// TIA Portal V19 export
TYPE "IF_TA2502"
TITLE = TA2502
// DEVICEID : 466
//  VENDOR : ifm electronic gmbh
//  DATE: 27.09.2021 
// 
//  Comment : Interface TA2502
   STRUCT
      StandardStructure : Struct
         Header : Struct
            NumberParameter : Int := 17;   // Number of device parameters (Device Identification + Device Parameter)
            AdressParamDownLoad : Int := 20;   // Start adress for ParamDownload signals in this struct
            AdressDeviceIndent : Int := 44;   // Start adress for Device Identification Parameters in this struct
            AdressApplicSpez : Int := 700;   // Start adress ApplicationSpezificTag
            AdressDeviceParam : Int := 782;   // Start adress for Device Parameters in this Area
            AdressKommando : Int := 942;   // Start adress for Device Commandos
            NumberCommandos : Int := 5;   // Number of Commandos of the device
            Spare01 : Int;   // spare
            Spare02 : Int;   // spare
            Spare03 : Int;   // spare
         END_STRUCT;
         Paramdownload : Struct
            ParamDownLoadStart : Struct   // Parameter Download Start (Only if master and device are V1.1)
               BlockStat : DWord;   // function block status
               IOLStat : DWord;   // IO-Link Status
            END_STRUCT;
            ParamDownLoadEnd : Struct   // Parameter Download End (Only if master and device are V1.1)
               BlockStat : DWord;   // function block status
               IOLStat : DWord;   // IO-Link Status
            END_STRUCT;
            ParamDownLoadStore : Struct   // Parameter Download Store (Only if master and device are V1.1)
               BlockStat : DWord;   // function block status
               IOLStat : DWord;   // IO-Link Status
            END_STRUCT;
         END_STRUCT;
         DeviceIndentification : Struct   // device indentification parameter
            V_VendorName : Struct   // Vendor Name
               Text : String[64];
               Index : Int := 16;   // parameter index
               Subindex : Int;   // parameter subindex
               Length : Int := 19;   // parameter length in BYTE for writing
               BlockStat : DWord;   // function block status
               IOLStat : DWord;   // IO-Link Status
               RelRead : Bool := TRUE;   // reading release
               RelWrite : Bool;   // writing release
            END_STRUCT;
            V_VendorText : Struct   // Vendor Text
               Text : String[64];
               Index : Int := 17;   // parameter index
               Subindex : Int;   // parameter subindex
               Length : Int := 11;   // parameter length in BYTE for writing
               BlockStat : DWord;   // function block status
               IOLStat : DWord;   // IO-Link Status
               RelRead : Bool := TRUE;   // reading release
               RelWrite : Bool;   // writing release
            END_STRUCT;
            V_ProductName : Struct   // Product Name
               Text : String[64];
               Index : Int := 18;   // parameter index
               Subindex : Int;   // parameter subindex
               Length : Int := 6;   // parameter length in BYTE for writing
               BlockStat : DWord;   // function block status
               IOLStat : DWord;   // IO-Link Status
               RelRead : Bool := TRUE;   // reading release
               RelWrite : Bool;   // writing release
            END_STRUCT;
            V_ProductID : Struct   // Product ID
               Text : String[64];
               Index : Int := 19;   // parameter index
               Subindex : Int;   // parameter subindex
               Length : Int := 6;   // parameter length in BYTE for writing
               BlockStat : DWord;   // function block status
               IOLStat : DWord;   // IO-Link Status
               RelRead : Bool := TRUE;   // reading release
               RelWrite : Bool;   // writing release
            END_STRUCT;
            V_ProductText : Struct   // Product Text
               Text : String[64];
               Index : Int := 20;   // parameter index
               Subindex : Int;   // parameter subindex
               Length : Int := 23;   // parameter length in BYTE for writing
               BlockStat : DWord;   // function block status
               IOLStat : DWord;   // IO-Link Status
               RelRead : Bool := TRUE;   // reading release
               RelWrite : Bool;   // writing release
            END_STRUCT;
            V_SerialNumber : Struct   // Serial Number
               Text : String[64];
               Index : Int := 21;   // parameter index
               Subindex : Int;   // parameter subindex
               Length : Int := 12;   // parameter length in BYTE for writing
               BlockStat : DWord;   // function block status
               IOLStat : DWord;   // IO-Link Status
               RelRead : Bool := TRUE;   // reading release
               RelWrite : Bool;   // writing release
            END_STRUCT;
            V_HardwareRevision : Struct   // Hardware Version
               Text : String[64];
               Index : Int := 22;   // parameter index
               Subindex : Int;   // parameter subindex
               Length : Int := 2;   // parameter length in BYTE for writing
               BlockStat : DWord;   // function block status
               IOLStat : DWord;   // IO-Link Status
               RelRead : Bool := TRUE;   // reading release
               RelWrite : Bool;   // writing release
            END_STRUCT;
            V_FirmwareRevision : Struct   // Firmware Version
               Text : String[64];
               Index : Int := 23;   // parameter index
               Subindex : Int;   // parameter subindex
               Length : Int := 5;   // parameter length in BYTE for writing
               BlockStat : DWord;   // function block status
               IOLStat : DWord;   // IO-Link Status
               RelRead : Bool := TRUE;   // reading release
               RelWrite : Bool;   // writing release
            END_STRUCT;
         END_STRUCT;
         ApplicationSpecificTag : Struct   // AppliciationSpecificTag
            V_ApplicationSpecificTa : Struct   // Application Specific Tag
               Text : String[64];
               Index : Int := 24;   // parameter index
               Subindex : Int;   // parameter subindex
               Length : Int := 16;   // parameter length in BYTE for writing
               BlockStat : DWord;   // function block status
               IOLStat : DWord;   // IO-Link Status
               RelRead : Bool := TRUE;   // reading release
               RelWrite : Bool := TRUE;   // writing release
            END_STRUCT;
         END_STRUCT;
         DeviceParameters : Struct   // Device Parameters
            Parameter_01 : Struct   // V_DeviceAccessLocks > Device Access Locks
               Value : Struct   // Parameter Value (must be always 4 Byte)
                  V_DeviceAccessLocks : Int;
                  Byte02 : Byte;
                  Byte03 : Byte;
               END_STRUCT;
               Index : Int := 12;   // parameter index
               Subindex : Int;   // parameter subindex
               Length : Int := 2;   // parameter length in BYTE for writing
               BlockStat : DWord;   // function block status
               IOLStat : DWord;   // IO-Link Status
               RelRead : Bool := TRUE;   // reading release
               RelWrite : Bool := TRUE;   // writing release
            END_STRUCT;
            Parameter_02 : Struct   // V_DeviceStatus > Device Status
               Value : Struct   // Parameter Value (must be always 4 Byte)
                  V_DeviceStatus : Byte;
                  Byte01 : Byte;
                  Byte02 : Byte;
                  Byte03 : Byte;
               END_STRUCT;
               Index : Int := 36;   // parameter index
               Subindex : Int;   // parameter subindex
               Length : Int := 1;   // parameter length in BYTE for writing
               BlockStat : DWord;   // function block status
               IOLStat : DWord;   // IO-Link Status
               RelRead : Bool := TRUE;   // reading release
               RelWrite : Bool;   // writing release
            END_STRUCT;
            Parameter_03 : Struct   // FOU2 > FOU2 [OUT 2] behaviour in case of fault
               Value : Struct   // Parameter Value (must be always 4 Byte)
                  FOU2 : Byte := BYTE#16#04;
                  Byte01 : Byte;
                  Byte02 : Byte;
                  Byte03 : Byte;
               END_STRUCT;
               Index : Int := 532;   // parameter index
               Subindex : Int;   // parameter subindex
               Length : Int := 1;   // parameter length in BYTE for writing
               BlockStat : DWord;   // function block status
               IOLStat : DWord;   // IO-Link Status
               RelRead : Bool := TRUE;   // reading release
               RelWrite : Bool := TRUE;   // writing release
            END_STRUCT;
            Parameter_04 : Struct   // uni > uni Selection of unit on the sensor display
               Value : Struct   // Parameter Value (must be always 4 Byte)
                  uni : Byte;
                  Byte01 : Byte;
                  Byte02 : Byte;
                  Byte03 : Byte;
               END_STRUCT;
               Index : Int := 551;   // parameter index
               Subindex : Int;   // parameter subindex
               Length : Int := 1;   // parameter length in BYTE for writing
               BlockStat : DWord;   // function block status
               IOLStat : DWord;   // IO-Link Status
               RelRead : Bool := TRUE;   // reading release
               RelWrite : Bool := TRUE;   // writing release
            END_STRUCT;
            Parameter_05 : Struct   // ou2 > ou2 Output configuration [OUT 2]
               Value : Struct   // Parameter Value (must be always 4 Byte)
                  ou2 : Byte := BYTE#16#01;
                  Byte01 : Byte;
                  Byte02 : Byte;
                  Byte03 : Byte;
               END_STRUCT;
               Index : Int := 590;   // parameter index
               Subindex : Int;   // parameter subindex
               Length : Int := 1;   // parameter length in BYTE for writing
               BlockStat : DWord;   // function block status
               IOLStat : DWord;   // IO-Link Status
               RelRead : Bool := TRUE;   // reading release
               RelWrite : Bool := TRUE;   // writing release
            END_STRUCT;
            Parameter_06 : Struct   // ASP2 > ASP2 Analogue start point 2. [ASP2] must be smaller than [AEP2]. Plea
               Value : Struct   // Parameter Value (must be always 4 Byte)
                  ASP2 : Int;
                  Byte02 : Byte;
                  Byte03 : Byte;
               END_STRUCT;
               Index : Int := 630;   // parameter index
               Subindex : Int;   // parameter subindex
               Length : Int := 2;   // parameter length in BYTE for writing
               BlockStat : DWord;   // function block status
               IOLStat : DWord;   // IO-Link Status
               RelRead : Bool := TRUE;   // reading release
               RelWrite : Bool := TRUE;   // writing release
            END_STRUCT;
            Parameter_07 : Struct   // AEP2 > AEP2 Analogue end point 2. [AEP2] must be greater than [ASP2]. Please
               Value : Struct   // Parameter Value (must be always 4 Byte)
                  AEP2 : Int := 2000;
                  Byte02 : Byte;
                  Byte03 : Byte;
               END_STRUCT;
               Index : Int := 631;   // parameter index
               Subindex : Int;   // parameter subindex
               Length : Int := 2;   // parameter length in BYTE for writing
               BlockStat : DWord;   // function block status
               IOLStat : DWord;   // IO-Link Status
               RelRead : Bool := TRUE;   // reading release
               RelWrite : Bool := TRUE;   // writing release
            END_STRUCT;
            Parameter_08 : Struct   // coF > coF Zero_point calibration (Calibration offset)
               Value : Struct   // Parameter Value (must be always 4 Byte)
                  coF : Int;
                  Byte02 : Byte;
                  Byte03 : Byte;
               END_STRUCT;
               Index : Int := 5001;   // parameter index
               Subindex : Int;   // parameter subindex
               Length : Int := 2;   // parameter length in BYTE for writing
               BlockStat : DWord;   // function block status
               IOLStat : DWord;   // IO-Link Status
               RelRead : Bool := TRUE;   // reading release
               RelWrite : Bool := TRUE;   // writing release
            END_STRUCT;
         END_STRUCT;
         Commando : Struct   // Commandos
            Commando_00 : Struct   // V_SystemCommand = Restore Factory Settings
               Value : Byte := BYTE#16#82;   // 2
               Index : Int := 2;   // parameter index
               Subindex : Int;   // parameter subindex
               Length : Int := 1;   // parameter length in BYTE for writing
               BlockStat : DWord;   // function block status
               IOLStat : DWord;   // IO-Link Status
            END_STRUCT;
            Commando_01 : Struct   // V_SystemCommand = IO_Link 1.1 system test command 240, Event 8DFE appears
               Value : Byte := BYTE#16#F0;   // 2
               Index : Int := 2;   // parameter index
               Subindex : Int;   // parameter subindex
               Length : Int := 1;   // parameter length in BYTE for writing
               BlockStat : DWord;   // function block status
               IOLStat : DWord;   // IO-Link Status
            END_STRUCT;
            Commando_02 : Struct   // V_SystemCommand = IO_Link 1.1 system test command 241, Event 8DFE disappears
               Value : Byte := BYTE#16#F1;   // 2
               Index : Int := 2;   // parameter index
               Subindex : Int;   // parameter subindex
               Length : Int := 1;   // parameter length in BYTE for writing
               BlockStat : DWord;   // function block status
               IOLStat : DWord;   // IO-Link Status
            END_STRUCT;
            Commando_03 : Struct   // V_SystemCommand = IO_Link 1.1 system test command 242, Event 8DFF appears
               Value : Byte := BYTE#16#F2;   // 2
               Index : Int := 2;   // parameter index
               Subindex : Int;   // parameter subindex
               Length : Int := 1;   // parameter length in BYTE for writing
               BlockStat : DWord;   // function block status
               IOLStat : DWord;   // IO-Link Status
            END_STRUCT;
            Commando_04 : Struct   // V_SystemCommand = IO_Link 1.1 system test command 243, Event 8DFF disappears
               Value : Byte := BYTE#16#F3;   // 2
               Index : Int := 2;   // parameter index
               Subindex : Int;   // parameter subindex
               Length : Int := 1;   // parameter length in BYTE for writing
               BlockStat : DWord;   // function block status
               IOLStat : DWord;   // IO-Link Status
            END_STRUCT;
         END_STRUCT;
      END_STRUCT;
   END_STRUCT;
END_TYPE
